PROGRAM MAIN
VAR
END_VAR

PRG_Camming();
FB_Servo1(CAMTABLE:=CAMTABLE , Axis:=Axis1 , Slave:=Axis2 , stAxisInterface:=AxisInterface1 );
FB_Servo2(CAMTABLE:=CAMTABLE , Axis:=Axis2 , Slave:=Axis1 , stAxisInterface:=AxisInterface2 );

END_PROGRAM

(* stored: Version 1.1.0.1, ProductVersion 3.1.4022.18
   POU MAIN: Id {c8d72e14-0a57-4650-8015-1b73cc590f1f}, SpecialFunc None *)
